FUNCTION_BLOCK TEST_BOOLN (* Test Boolean NAND,NOR *)
  (* Standard: 61499-1 *)
  (* Version 0.0, 2006-09-19, JHC, Holobloc Inc *)
  (* Compiler header: package fb.rt.test; *)
  (* Compiler classdef: SimpleFB *)
  (* Compiler Java Sun JDK 1.5.0 *)
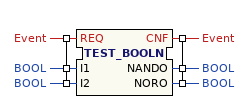
  EVENT_INPUT
    REQ WITH I1, I2;
  END_EVENT
  EVENT_OUTPUT
    CNF WITH NANDO, NORO;
  END_EVENT
  VAR_INPUT
    I1 : BOOL;
    I2 : BOOL;
  END_VAR
  VAR_OUTPUT
    NANDO : BOOL;
    NORO : BOOL;
  END_VAR
  ALGORITHM REQ IN FBD:
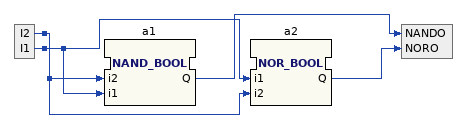
    FBS
      a1 : NAND_BOOL;
      a2 : NOR_BOOL;
    END_FBS
    DATA_CONNECTIONS
      I2 TO a1.i2;
      I1 TO a2.i1;
      I1 TO a1.i1;
      a1.Q TO NANDO;
      I2 TO a2.i2;
      a2.Q TO NORO;
    END_CONNECTIONS
  END_ALGORITHM
END_FUNCTION_BLOCK
